(* PLC project Senza_nome, Sconosciuto Senza_nome 1 *)
(* stored: creationDateTime 2026-08-24T13:36:20, modificationDateTime 2026-08-24T13:47:10 *)

PROGRAM program0
  VAR
    CTU0 : CTU;
  END_VAR
  VAR
    BT1 AT %IX100.0 : BOOL;
    BT2 AT %IX100.1 : BOOL;
    Led AT %QX100.0 : BOOL;
  END_VAR
  VAR
    PV : INT := 5;
  END_VAR
  VAR  (* added by the conversion: wires and edge detectors of the diagram *)
    R_TRIG1 : R_TRIG;
  END_VAR

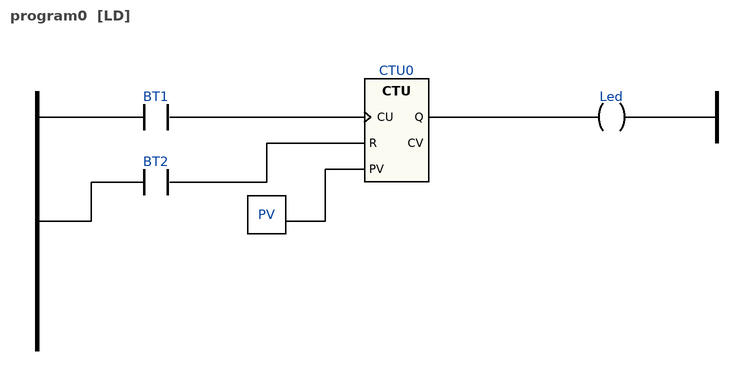
(* LD diagram, written out as Structured Text *)
R_TRIG1(CLK := BT1);
CTU0(CU := R_TRIG1.Q, R := BT2, PV := PV);
Led := CTU0.Q;
END_PROGRAM

CONFIGURATION Config0
  RESOURCE Res0 ON PLC
    TASK task0(INTERVAL := T#20ms, PRIORITY := 0);
    PROGRAM instance0 WITH task0 : program0;
  END_RESOURCE
END_CONFIGURATION
